FUNCTION A_DATE : ST_Arg
VAR_INPUT
	obj	: REFERENCE TO DATE;
END_VAR

IF __ISVALIDREF(obj) THEN
	A_DATE.eType := E_ArgType.DateArg;
	A_DATE.pData := ADR(obj);
	A_DATE.nSize := SIZEOF(DATE);
END_IF

END_FUNCTION

(* stored: Version 1.1.0.1, ProductVersion 3.1.4024.15
   POU A_DATE: Id {fbb3fe98-7bfe-4c88-9997-57e3b7cfe99c}, SpecialFunc None *)
